FUNCTION_BLOCK FB_EL3453_handling
VAR_INPUT
END_VAR
VAR_OUTPUT
END_VAR
VAR
END_VAR

END_FUNCTION_BLOCK

(* stored: Version 1.1.0.1, ProductVersion 3.1.4024.11
   POU FB_EL3453_handling: Id {607e69df-f40a-48cc-8fb1-54e07d0aad99}, SpecialFunc None *)
